PROGRAM CountPosition
VAR
END_VAR

IF IO.StepRotatonSwitch = 1 AND IO.Initialized THEN
		IO.LEDGreen := 0;
		IF IO.MotorRotationDirection = 0 THEN
			IF IO.MotorRotation = 1 OR NOT IO.Switch AND Automatic.RotationPositionCurrent < 190 THEN
				Automatic.RotationPositionCurrent := Automatic.RotationPositionCurrent + 1;
			END_IF
			//IF NOT IO.Switch THEN
			//	Automatic.RotationPositionAuto := Automatic.RotationPositionAuto + 1;
			//END_IF
		ELSE
			IF IO.MotorRotation = 1 OR NOT IO.Switch AND NOT IO.EndRotationSensor THEN
				Automatic.RotationPositionCurrent := Automatic.RotationPositionCurrent - 1;
			END_IF
			//IF NOT IO.Switch THEN
			//	Automatic.RotationPositionAuto := Automatic.RotationPositionAuto - 1;
			//END_IF
		END_IF
	ELSE
		IO.LEDGreen := 1;
	END_IF
	
	IF IO.StepExtensionSwitch = 1 AND IO.Initialized THEN
		IO.LEDGreen := 0;
		IF IO.MotorExtensionDirection = 0 THEN
			IF IO.MotorExtension OR NOT IO.Switch AND Automatic.ExtensionPositionCurrent < 388 THEN
				Automatic.ExtensionPositionCurrent := Automatic.ExtensionPositionCurrent + 1;
			END_IF
			//IF NOT IO.Switch THEN
			//	Automatic.ExtensionPositionAuto := Automatic.ExtensionPositionAuto + 1;
			//END_IF
		ELSE
			IF IO.MotorExtension OR NOT IO.Switch AND NOT IO.EndExtensionSensor THEN
				Automatic.ExtensionPositionCurrent := Automatic.ExtensionPositionCurrent - 1;
			END_IF
			//IF NOT IO.Switch THEN
			//	Automatic.ExtensionPositionAuto := Automatic.ExtensionPositionAuto - 1;
			//END_IF
		END_IF
	ELSE
		IO.LEDGreen := 1;
	END_IF
	
	IF IO.StepLiftingSwitch = 1 AND IO.Initialized THEN
		IO.LEDGreen := 0;
		IF IO.MotorLiftingDirection = 0 THEN
			IF IO.MotorLifting OR NOT IO.Switch THEN
				Automatic.LiftingPositionCurrent := Automatic.LiftingPositionCurrent + 1;
			END_IF
			//IF NOT IO.Switch THEN
			//	Automatic.LiftingPositionAuto := Automatic.LiftingPositionAuto + 1;
			//END_IF
		ELSE
			IF IO.MotorLifting OR NOT IO.Switch AND NOT IO.EndLiftingSensor THEN
				Automatic.LiftingPositionCurrent := Automatic.LiftingPositionCurrent - 1;
			END_IF
			//IF NOT IO.Switch THEN
			//	Automatic.LiftingPositionAuto := Automatic.LiftingPositionAuto - 1;
			//END_IF
		END_IF
	ELSE
		IO.LEDGreen := 1;
	END_IF
	IF IO.StepGripSwitch = 1 AND IO.Initialized THEN	// inverted
		IO.LEDGreen := 0;
		IF IO.MotorGripDirection = 0 THEN
			IF IO.MotorGrip OR NOT IO.Switch AND Automatic.GripPositionCurrent < 80 THEN
				Automatic.GripPositionCurrent := Automatic.GripPositionCurrent + 1;
			END_IF
			//IF NOT IO.Switch THEN
			//	Automatic.GripPositionAuto := Automatic.GripPositionAuto + 1;
			//END_IF
		ELSE
			IF IO.MotorGrip OR NOT IO.Switch AND NOT IO.EndGripSensor THEN
				Automatic.GripPositionCurrent := Automatic.GripPositionCurrent - 1;
			END_IF
			//IF NOT IO.Switch THEN
			//	Automatic.GripPositionAuto := Automatic.GripPositionAuto - 1;
			//END_IF
		END_IF
	ELSE
		IO.LEDGreen := 1;
	END_IF

END_PROGRAM

(* stored: Version 1.1.0.1, ProductVersion 3.1.4024.13
   POU CountPosition: Id {66a3fea9-06ea-4e58-ba00-8e91517712ea}, SpecialFunc None *)
